DATA_BLOCK "R_TRIG_DB_1"
{InstructionName := 'R_TRIG';
 LibVersion := '1.0';
 S7_Optimized_Access := 'TRUE' }
AUTHOR : SIMATIC
FAMILY : BIT
NAME : R_TRIG
VERSION : 1.0
NON_RETAIN
R_TRIG

BEGIN

END_DATA_BLOCK

